FUNCTION F_SerialCrc16 : WORD
VAR_INPUT
    pData   : POINTER TO BYTE;
    nLength : UINT;
END_VAR
VAR
    nByte : UINT;
    nBit  : INT;
    wCrc  : WORD := 16#FFFF;
END_VAR

wCrc := 16#FFFF;

IF (pData = 0) OR (nLength = 0) THEN
    F_SerialCrc16 := wCrc;
    RETURN;
END_IF;

FOR nByte := 0 TO nLength - 1 DO
    wCrc := wCrc XOR BYTE_TO_WORD(pData[nByte]);

    FOR nBit := 0 TO 7 DO
        IF (wCrc AND 16#0001) <> 0 THEN
            wCrc := SHR(wCrc, 1) XOR 16#A001;
        ELSE
            wCrc := SHR(wCrc, 1);
        END_IF;
    END_FOR;
END_FOR;

F_SerialCrc16 := wCrc;

END_FUNCTION

(* stored: Version 1.1.0.1, ProductVersion 3.1.4026.20
   POU F_SerialCrc16: Id {8D8FD1C5-6CC1-4111-B330-5478FCD6DAC6}, SpecialFunc None *)
